Staubli VAL3: goHome.pgx

program goHome()
begin
  // go to HOME
  waitEndMove()

  cycleStatus:bToHome=true
  //

end
